FUNCTION_BLOCK FB_LoggerFactory IMPLEMENTS I_Logger
VAR
	fbList:						FB_ListLogger;
	nIndex: 					DINT;
	nEvent:						DINT;
	nLength:					DINT;
	pEvent:						POINTER TO ST_Event;	
END_VAR

// Provide the Logging function to a module, and event buffer
// Hmi anyway have to work with a static list :-(

// Deactivate old events
nIndex:= 0;
WHILE nIndex < nLength DO
	IF pEvent[nIndex].Active AND pEvent[nIndex].EventType <> E_Event.Error THEN
		pEvent[nIndex].Active:= FALSE;
	ELSE
		M_Remove(nIndex);		
	END_IF
	nIndex := nIndex + 1;
END_WHILE

METHOD FB_init : BOOL
VAR_INPUT
	bInitRetains : BOOL; // if TRUE, the retain variables are initialized (warm start / cold start)
	bInCopyCode : BOOL;  // if TRUE, the instance afterwards gets moved into the copy code (online change)
	pEvent:						POINTER TO ST_Event;
	nEvent:						DINT;
END_VAR
THIS^.pEvent:= pEvent;
THIS^.nEvent:= nEvent;
END_METHOD

METHOD PUBLIC M_Attach
VAR_INPUT
	Logger:		I_Logger;
END_VAR
// Attach
fbList.M_Add(Logger);
END_METHOD

METHOD PUBLIC M_Dettach
VAR_INPUT
	Logger:		I_Logger;
END_VAR
// Attach
fbList.M_Remove(Logger);
END_METHOD

METHOD PUBLIC M_Find : DINT
VAR_INPUT
	stEvent:	ST_Event;
END_VAR
M_Find := -1;
nIndex:= 0;
WHILE nIndex < nLength DO
	IF (pEvent[nIndex].Source = stEvent.Source) AND_THEN
    	(pEvent[nIndex].EventType = stEvent.EventType) AND_THEN
		(pEvent[nIndex].Instance = stEvent.Instance) AND_THEN
		(pEvent[nIndex].Class = stEvent.Class) AND_THEN
		(pEvent[nIndex].Message = stEvent.Message) THEN
        M_Find := nIndex;
        RETURN;
    END_IF
	nIndex := nIndex + 1;
END_WHILE
END_METHOD

METHOD PUBLIC M_Log
VAR_INPUT
	stEvent:		ST_Event;
END_VAR
IF (nIndex:=  M_Find(stEvent)) >= 0 THEN
	// Update existing eventss
	pEvent[nIndex].Active:= TRUE;
	pEvent[nIndex].Arguments:= stEvent.Arguments;
ELSE
	// add new event
	stEvent.Active:= TRUE;
	M_Publish(stEvent);
	pEvent[nLength]:= stEvent;
	nLength:= nLength + 1;
END_IF
END_METHOD

METHOD M_Publish
VAR_INPUT
	stEvent:	ST_Event;
END_VAR
// Publis new events
nIndex:= 0;
WHILE nIndex < fbList.P_Length DO
	fbList.M_Index(nIndex).M_Log(stEvent);
	nIndex := nIndex + 1;
END_WHILE
END_METHOD

METHOD PUBLIC M_Remove : Bool
VAR_INPUT
	Index:		DINT;
END_VAR
// Remove event
MEMCPY(ADR(pEvent[Index]), ADR(pEvent[Index + 1]), SIZEOF(ST_Event) * DINT_TO_UDINT(nEvent - nLength));
nLength:= nLength - 1;
END_METHOD

METHOD PUBLIC M_Reset
VAR_INPUT
END_VAR
// Reset Errors
nIndex:= 0;
WHILE nIndex < nLength DO
	IF pEvent[nIndex].EventType = E_Event.Error THEN
		M_Remove(nIndex);
	END_IF
	nIndex := nIndex + 1;
END_WHILE
END_METHOD

END_FUNCTION_BLOCK

(* stored: Version 1.1.0.1
   POU FB_LoggerFactory: Id {14a5296c-b52d-02f9-2d9e-abab1d7b93f2}, SpecialFunc None
   Method FB_init: Id {6df5be79-0a0c-0d2a-0a65-cf7790a42dfd}
   Method M_Attach: Id {85d5015d-7e39-4cfd-a721-66b108eef110}
   Method M_Dettach: Id {693d57be-522c-4fd2-923e-e39bc4f52f84}
   Method M_Find: Id {57ee7645-77de-477e-aa71-8b5ff862f016}
   Method M_Log: Id {970a1cce-913f-4f52-a720-54d7dfe3d1a3}
   Method M_Publish: Id {578d5b47-6fac-0518-1a61-62b0162be35c}
   Method M_Remove: Id {a03dc35c-ef8e-043d-3adb-f11c8fb4c08b}
   Method M_Reset: Id {9e416491-698f-0c93-2f87-8032ff6306d1} *)
